// TwinCAT 3 PLC project PLC
// Title: CNC Sample Code using Tria-Link
// Company: Triamec Motion AG
// Author: Triamec Motion AG
// Description: CNC Sample Code using Tria-Link
// ProgramVersion: 3.1.4024.0
// libraries:
//   Tc2_CncHli, * (Beckhoff Automation GmbH)
//   Tc2_Standard, * (Beckhoff Automation GmbH)
//   Tc2_System, * (Beckhoff Automation GmbH)
//   Tc3_Module, * (Beckhoff Automation GmbH)
//   Triamec, * (Triamec Motion AG)
// project tree:
//   / Fast_Task.TcTTO, Slow_Task.TcTTO
//   POUs/ Triamec_GVL.TcGVL (not stored), MAIN.TcPOU, MAIN_FAST.TcPOU, CNC_Axis.TcPOU
// real-time tasks:
//   TASK Slow_Task: cycle T#10ms, priority 12, ADS port 350
// I/O:
//   DEVICE TriaLink (NOV-DP-RAM)
//   DEVICE Sercos (FC75xx) (disabled)
//     Drive 1 (Sercos Drive)
//     Drive 2 (Sercos Drive)
// variable links:
//   PLC/PLC Instance <-> CNC/Axes/Axis_1
//     Fast_Task Inputs/MAIN.Axes[1].SercosPosCmd <-> Outputs/Position command value
//     Fast_Task Outputs/MAIN.Axes[1].SercosPosAct <-> Inputs/Position feedback 1 value
//     Slow_Task Outputs/MAIN.Axes[1].SercosPhase <-> Inputs/Sercos Phase
//     Slow_Task Outputs/MAIN.Axes[1].SercosStatus <-> Inputs/Drive status word
//   PLC/PLC Instance <-> CNC/Axes/Axis_2
//     Fast_Task Inputs/MAIN.Axes[2].SercosPosCmd <-> Outputs/Position command value
//     Fast_Task Outputs/MAIN.Axes[2].SercosPosAct <-> Inputs/Position feedback 1 value
//     Slow_Task Outputs/MAIN.Axes[2].SercosPhase <-> Inputs/Sercos Phase
//     Slow_Task Outputs/MAIN.Axes[2].SercosStatus <-> Inputs/Drive status word

CONFIGURATION PLC
    RESOURCE PLC ON TwinCAT3
        TASK Fast_Task(INTERVAL := T#1ms, PRIORITY := 4);
        TASK Slow_Task(INTERVAL := T#10ms, PRIORITY := 12);
        PROGRAM MAIN_FAST WITH Fast_Task : MAIN_FAST;
        PROGRAM MAIN WITH Slow_Task : MAIN;
    END_RESOURCE
END_CONFIGURATION

// ---- POUs/MAIN_FAST.TcPOU
PROGRAM MAIN_FAST
VAR
	i : USINT; (* counter variable *)
END_VAR

(* --------------------------------------------- *)
(* Triamec Motion AG, 6340 Baar, Switzerland     *)
(* Sample Code may be adapted to customer need   *)
(* --------------------------------------------- *)

(* Tria-Link cyclic fast call *)
MAIN.Trialink.CallFast();

(* CNC axis cyclic fast call *)
FOR i := 1 TO MAIN.cAxes DO
	MAIN.Axes[i].Fast();
END_FOR

END_PROGRAM

// ---- POUs/MAIN.TcPOU
PROGRAM MAIN
VAR CONSTANT
	cAxes			: USINT := 2; (* Number of axes in use *)
END_VAR

VAR
	Trialink : Triamec.TL_Trialink2; 			(* the Tria-Link adapter *)
	Hli	: MCV_HliInterface; 					(* Hli interface *)
	Axes : ARRAY [1..cAxes] OF CNC_Axis; 	(* the extended triamec axis object with link to the CNC *)
	
	initDone : BOOL;	(* initialization done *)
	i : USINT; 			(* counter variable *)
END_VAR

(* ------------------------------------------- *)
(* Triamec Motion AG, 6340 Baar, Switzerland   *)
(* Sample Code may be adapted to customer need *)
(* ------------------------------------------- *)

(* Tria-Link and Axes configuration *)
IF NOT initDone THEN
	initDone := Config();
END_IF

(* Tria-Link cyclic call*)
Trialink.Execute := gEnableTrialink;
Trialink.CallSlow();
gCommunicationReady := gEnableTrialink AND NOT Trialink.Error;

(* HLI interface *)
IF NOT Hli.Initialized THEN
	Hli(); // initialize HLI
END_IF

(* Axes cyclic call *)
FOR i := 1 TO cAxes DO
	Axes[i].iAxis := i;				// logical axis number
	Axes[i].reset := gResetAxes; 	// reset drive errors
	Axes[i].enable := gEnableAxes; 	// set enable / disable
	Axes[i].couple := TRUE;			// couple drive to CNC pathplanner
	Axes[i](Hli := Hli, Trialink := Trialink); 	// cyclic call of cnc axes
	gCommunicationReady	:= gCommunicationReady AND Axes[i].ready;
END_FOR

METHOD Config : BOOL
(* Tria-Link configuration *)
Trialink.Config.nDevId := 1; // NOV-DP-RAM Id, see TwinCAT System Manager (I/0 > Devices > TriaLink) 
Trialink.Config.TcEventEnable := TRUE;

(* Axes configuration *)
(* ---------- Axis 1 ---------- *)
Axes[1].inc_per_unit 		:= 1000000; // scale between CNC and PLC
Axes[1].Config.Simulate   	:= FALSE;
Axes[1].Config.Station    	:= 10;		// The drive address
Axes[1].Config.SubAxis    	:= TL_Config.SubAxis.FirstAxis; // first or second axis of a two axes drive
Axes[1].Config.GearFactor 	:= 1;		// multiplication factor of position and velocity data
Axes[1].Config.ModuloWrap 	:= 0;		// modulo wrap for rotation axes
Axes[1].referencePos 		:= 0.0;		// reference position to which the axis is set after homing
	
(* ---------- Axis 2 ---------- *)
Axes[2].inc_per_unit 		:= 1000000; // scale between CNC and PLC
Axes[2].Config.Simulate   	:= TRUE;
Axes[2].Config.Station    	:= 10;		// The drive address
Axes[2].Config.SubAxis    	:= TL_Config.SubAxis.SecondAxis; // first or second axis of a two axes drive
Axes[2].Config.GearFactor 	:= 1;		// multiplication factor of position and velocity data
Axes[2].Config.ModuloWrap 	:= 0;		// modulo wrap for rotation axes
Axes[2].referencePos 		:= 0.0; 	// reference position to which the axis is set after homing

Config := TRUE;
END_METHOD

END_PROGRAM

// ---- POUs/CNC_Axis.TcPOU
FUNCTION_BLOCK CNC_Axis EXTENDS Triamec.TL_Axis2
VAR_IN_OUT
	Trialink	: Triamec.TL_Trialink2; (* the Tria-Link adapter *)
	Hli			: MCV_HliInterface; (* HLI interface *)
END_VAR
VAR_INPUT
	inc_per_unit : LREAL := 1E7; (* use 10000 inc/deg or 1E7 inc/m *)
END_VAR
VAR_OUTPUT
	messageString  : STRING(100); (* error message *)
END_VAR
VAR
	SercosPhase AT %Q*	: WORD; (* CNC > GEO > Axis > Inputs > Sercos Phase *)
	SercosStatus AT %Q*	: WORD; (* CNC > GEO > Axis > Inputs > Drive status word *)
	SercosPosCmd AT %I*	: DINT; (* CNC > GEO > Axis > Outputs > Position command value *) 
	SercosPosAct AT %Q*	: DINT; (* CNC > GEO > Axis > Inputs > Position feedback 1 value *)		
	
	MessageHandler	: TL_AxisMessageHandler;	// provides corresponding message string
	TcEventLib		: TL_TwinCatError;
	TcEventDrv		: TL_TwinCatError;
END_VAR

(* --------------------------------------------- *)
(* Triamec Motion AG, 6340 Baar, Switzerland     *)
(* Sample Code may be adapted to customer need   *)
(* --------------------------------------------- *)

(* 
	we do not want any offset beween drive and cnc 
    because the drives have there own setPosition
	therefore set the following parameters in the axis of the cnc:
		kenngr.abs_pos_gueltig			1
		kenngr.set_refpos_mode         	OFFSET
		kenngr.set_refpos_offset		0
	this mode ensures, that the cnc does not set cmdPos=actPos when
	MCControlBoolUnit_SetReferencePosition is set
*)

SUPER^.CallSlow(Trialink := THIS^.Trialink);

// CNC axis handler
IF Hli.Initialized AND iAxis >= 1 AND HLI_SYS_AX_MaxIdx >= iAxis THEN
	(* enable plc control for axis *)
	gpAx[iAxis-1]^.head.plc_present_w := TRUE;
	
	(* enable PLC to drive HLI interface *)
	gpAx[iAxis-1]^.lr_mc_control.torque_permission.enable_w			:= TRUE;
	gpAx[iAxis-1]^.lr_mc_control.release_feedhold.enable_w 			:= TRUE;
	gpAx[iAxis-1]^.lr_mc_control.drive_on.enable_w 					:= TRUE;
	gpAx[iAxis-1]^.lr_mc_control.set_reference_position.enable_w	:= TRUE;
	gpAx[iAxis-1]^.lr_mc_control.follow_up.enable_w 				:= TRUE;
	
	(* set regulation and feed *)
	gpAx[iAxis-1]^.lr_mc_control.torque_permission.command_w		:= coupled;
	gpAx[iAxis-1]^.lr_mc_control.release_feedhold.command_w 		:= enabled;
	gpAx[iAxis-1]^.lr_mc_control.drive_on.command_w 				:= ready;
	
	(* Sercos interface	to CNC *)		
	sercosPhase	:= 4 * BOOL_TO_WORD(ready);
	sercosStatus:=   16#8000 * BOOL_TO_WORD(enabled)
						+ 16#4000 * BOOL_TO_WORD(coupled OR (ready AND NOT(enabled)))
						+ 16#2000 * BOOL_TO_WORD(error);
						
						
	(* The axis is set to tracking operation (follow up) on or off, i.e. the control loop is opened. The command position implicitly is set to the actual position. *)
	gpAx[iAxis-1]^.lr_mc_control.follow_up.command_w := followMe;
	
	(* HomingPosition *)
	gpAx[iAxis-1]^.lr_mc_control.set_reference_position.command_w	:= referenced;
END_IF

// This reads the drive message string into messageHandler.messageString and then sets messageHandler.done
messageHandler.execute := messageId >= TL_Message.Error; // show only errors
messageHandler(axis:=MC_axis, Trialink:=THIS^.Trialink);

// This generates a TwinCAT event in case of an axis library error and an axis drive error
TcEventLib.Execute	:= THIS^.Trialink.Done AND NOT (THIS^.Trialink.Error OR MC_axis.simulate);
TcEventLib.errorId	:= MC_axis.errorId;
TcEventLib.source	:= TL_EventSourceId.AxisLib; // See source entry in file triamecEventsTrialink.xml
TcEventLib.par1		:= MC_axis.iAxis;
TcEventLib();

TcEventDrv.Execute	:= TcEventLib.Execute AND MC_axis.messageId>=TL_Message.Error; // show only errors 
TcEventDrv.errorId	:= MC_axis.messageId;
TcEventDrv.source	:= TL_EventSourceId.AxisDrive; // See source entry in the file triamecEventsDrive.xml
TcEventDrv.par1		:= MC_axis.iAxis;
TcEventDrv();

METHOD Fast
VAR
	positionAct : LREAL; (* actual position *)
END_VAR
// The warning can be disabled here as the user is aware of the risk that the reference may not be valid by checking its validity
{warning disable C0371}

// Checking the VAR_IN_OUT reference, leave the current method in case of invalid reference
IF NOT __ISVALIDREF(Trialink) THEN
     RETURN;
END_IF

(* get the coordinates from the NC/CNC and write it to the drive *)
fastPositionCmd := DINT_TO_LREAL( SercosPosCmd ) / inc_per_unit;
SUPER^.CallFast( Trialink := Trialink );

(* get the actual position from the drive and pass it to NC *)
positionAct := ActualPositionFast(Trialink := Trialink);
(* coerse position to DINT range *)
IF ABS(positionAct * inc_per_unit) < 16#7FFFFFFF  THEN
	SercosPosAct := LREAL_TO_DINT(positionAct * inc_per_unit);
ELSIF positionAct < 0 THEN
	SercosPosAct := TO_DINT(16#80000000);
ELSE
	SercosPosAct := 16#7FFFFFFF;
END_IF

// The warning may be restored at the end of the access area
{warning restore C0371}
END_METHOD

END_FUNCTION_BLOCK
